// TIA Portal project "Energy_Monitoring_Project" (V17)

(* hardware
DEVICE "S7-1200 station_1"  S7-1200 Station
   slot 0: "Rack_0"  S7-1200 Rack  Rack  V1.0
   slot 1: "PLC_1"  CPU 1214C DC/DC/DC  6ES7 214-1AG40-0XB0  V4.5
DEVICE "HMI_1"  TP700 Comfort
   slot 0: "HMI_1"  TP700 Comfort  6AV2 124-0GC01-0AX0  17.0.0.0
   slot 1: "HMI_RT_1"  TP700 Comfort  6AV2 124-0GC01-0AX0  17.0.0.0
   slot 5: "HMI_1.IE_CP_1"  PROFINET Interface  17.0.0.0
      slot 1: "PROFINET Interface_1"  PROFINET Interface
         slot 1: "Port_1"  Port
         slot 2: "Port_2"  Port
   slot 7: "HMI_1.MPI/DP_CP_1"  MPI/DP Interface  17.0.0.0
*)

// ===== PLC "PLC_1"  CPU 1214C DC/DC/DC =====

VAR_GLOBAL   // PLC tag table "Default tag table"
   "Tag_1" AT %MW0 : Word;
   "Tag_2" AT %MW2 : Word;
   "Tag_3" AT %MW4 : Word;
   "Tag_4" AT %MW6 : Word;
   "Tag_5" AT %MW8 : Word;
   "Tag_6" AT %MW10 : Word;
   "Tag_7" AT %MW12 : Word;
   "Tag_8" AT %MW14 : Word;
   "Tag_9" AT %MW16 : Word;
END_VAR

DATA_BLOCK "Zone1_DB"   // DB1
{ S7_Optimized_Access := 'TRUE' }
VERSION : 0.1
   VAR
      Voltage : Real;
      Current : Real;
      kW : Real;
      kWh : Real;
      Threshold_Exceeded : Bool;
   END_VAR
BEGIN
END_DATA_BLOCK

DATA_BLOCK "Zone2_DB"   // DB2
{ S7_Optimized_Access := 'TRUE' }
VERSION : 0.1
   VAR
      Voltage : Real;
      Current : Real;
      kW : Real;
      kWh : Real;
      Threshold_Exceeded : Bool;
   END_VAR
BEGIN
END_DATA_BLOCK

DATA_BLOCK "Zone3_DB"   // DB3
{ S7_Optimized_Access := 'TRUE' }
VERSION : 0.1
   VAR
      Voltage : Real;
      Current : Real;
      kW : Real;
      kWh : Real;
      Threshold_Exceeded : Bool;
   END_VAR
BEGIN
END_DATA_BLOCK

DATA_BLOCK "Config_DB"   // DB4
{ S7_Optimized_Access := 'TRUE' }
VERSION : 0.1
   VAR
      Zone1_Threshold : Real := 50.0;   // Zone 1 max kW
      Zone2_Threshold : Real := 30.0;   // Zone 2 max kW
      Zone3_Threshold : Real := 20.0;   // Zone 3 max kW
      Total_Threshold : Real := 90.0;   // Total plant nax kW
      Shift_Start_Hour : Int := 8;   // Shift start time
      Alert_Enabled : Bool := true;   // Enable alerts
      Total_Power : Real;   // Total Power
      Shift_Number : Int := 1;
      Shift_Start_KWh : Real;
      Shift_Consumption : Real;
   END_VAR
BEGIN
END_DATA_BLOCK

DATA_BLOCK "Alarm_DB"   // DB5
{ S7_Optimized_Access := 'TRUE' }
VERSION : 0.1
   VAR
      Total_Exceeded : Bool;
      Alarm_Word : Word;
      Zone1_Alarm : Bool;
      Zone2_Alarm : Bool;
      Zone3_Alarm : Bool;
      Any_Alarm : Bool;
   END_VAR
BEGIN
END_DATA_BLOCK

DATA_BLOCK "Zone1_Reader_DB"   // DB6
{ S7_Optimized_Access := 'TRUE' }
VERSION : 0.1
// stored: InstanceOfName FB1_Energy_Reader
"FB1_Energy_Reader"
BEGIN
END_DATA_BLOCK

DATA_BLOCK "Zone2_Reader_DB"   // DB7
{ S7_Optimized_Access := 'TRUE' }
VERSION : 0.1
// stored: InstanceOfName FB1_Energy_Reader
"FB1_Energy_Reader"
BEGIN
END_DATA_BLOCK

DATA_BLOCK "Zone3_Reader_DB"   // DB8
{ S7_Optimized_Access := 'TRUE' }
VERSION : 0.1
// stored: InstanceOfName FB1_Energy_Reader
"FB1_Energy_Reader"
BEGIN
END_DATA_BLOCK

FUNCTION_BLOCK "FB1_Energy_Reader"   // FB1, SCL
{ S7_Optimized_Access := 'TRUE' }
VERSION : 0.1
   VAR_INPUT
      Voltage_Raw : Int;   // Raw analog voltage
      Current_Raw : Int;   // Raw analog current
      Power_Raw : Int;   // Raw analog power
      Zone_Name : String;   // Zone identifier
      Power_Threshold : Real;   // Alert thershold kW
   END_VAR
   VAR_OUTPUT
      Voltage : Real;   // Actual voltage V
      Current : Real;   // Actual Current A
      Active_Power : Real;   // Active Power kW
      Energy_kWh : Real;   // Cumulative energy
      Threshold_Exceeded : Bool;   // Alert flag
      Power_Factor : Real;   // PF calculation
   END_VAR
   VAR
      last_Power : Real;   // Previous scan power
      Scan_Timer : TON_TIME;   // 1 second timer
      kWh_Accumulator : Real;   // Running total
   END_VAR
BEGIN
   // --- Scale analog inputs ---
   #Voltage := INT_TO_REAL(#Voltage_Raw) / 27648.0 * 415.0;
   #Current := INT_TO_REAL(#Current_Raw) / 27648.0 * 100.0;
   #Active_Power := (#Voltage * #Current * #Power_Factor) / 1000.0;

   // --- Calculate kWh every second ---
   #Scan_Timer(IN := TRUE,
               PT := T#1S);

   IF #Scan_Timer.Q THEN
       #kWh_Accumulator := #kWh_Accumulator + (#Active_Power / 3600.0);
       #Scan_Timer(IN := FALSE,
                   PT := T#1S);
   END_IF;

   #Energy_kWh := #kWh_Accumulator;

   // --- Threshold check ---
   #Threshold_Exceeded := #Active_Power > #Power_Threshold;

   // --- Power factor (simplified) ---
   IF #Voltage > 0.0 AND #Current > 0.0 THEN
       #Power_Factor := 0.85; // Default - real system uses meter register
   END_IF;
END_FUNCTION_BLOCK

FUNCTION "FC1_Power_Calculation" : Void   // FC1, SCL
{ S7_Optimized_Access := 'TRUE' }
VERSION : 0.1
BEGIN
END_FUNCTION

FUNCTION "FC2_Alarm_generator" : Void   // FC2, SCL
{ S7_Optimized_Access := 'TRUE' }
VERSION : 0.1
   VAR_INPUT
      Zone1_Exceeded : Bool;
      Zone2_Exceeded : Bool;
      Zone3_Exceeded : Bool;
      Total_Exceeded : Bool;
   END_VAR
   VAR_OUTPUT
      Alarm_Word : Word;
      Any_Alarm : Bool;
   END_VAR
BEGIN
   // Pack alarms into word bits
   #Alarm_Word.%X0 := #Zone1_Exceeded;
   #Alarm_Word.%X1 := #Zone2_Exceeded;
   #Alarm_Word.%X2 := #Zone3_Exceeded;
   #Alarm_Word.%X3 := #Total_Exceeded;

   //Any alarm active
   #Any_Alarm := #Zone1_Exceeded OR
                 #Zone2_Exceeded OR
                 #Zone3_Exceeded OR
                 #Total_Exceeded;
END_FUNCTION

ORGANIZATION_BLOCK "Main"   // OB1, SCL, ProgramCycle
TITLE = "Main Program Sweep (Cycle)"
{ S7_Optimized_Access := 'TRUE' }
VERSION : 0.1
   VAR_INPUT
      Initial_Call : Bool;   // Initial call of this OB
      Remanence : Bool;   // =True, if remanent data are available
   END_VAR
BEGIN
   // ═══ ENERGY MONITORING SYSTEM ═══

   // Zone 1 — popup will ask to create Zone1_Reader_DB
   "Zone1_Reader_DB"(
                     Voltage_Raw     := "Tag_1",
                     Current_Raw     := "Tag_2",
                     Power_Raw       := "Tag_3",
                     Power_Threshold := "Config_DB".Zone1_Threshold);

   "Zone1_DB".kWh := "Zone1_Reader_DB".Energy_kWh;
   "Zone1_DB".kW := "Zone1_Reader_DB".Active_Power;

   // Zone 2
   "Zone2_Reader_DB"(
                     Voltage_Raw     := "Tag_4",
                     Current_Raw     := "Tag_5",
                     Power_Raw       := "Tag_6",
                     Power_Threshold := "Config_DB".Zone2_Threshold);

   "Zone2_DB".kWh := "Zone2_Reader_DB".Energy_kWh;
   "Zone2_DB".kW := "Zone2_Reader_DB".Active_Power;

   // Zone 3
   "Zone3_Reader_DB"(
                     Voltage_Raw     := "Tag_7",
                     Current_Raw     := "Tag_8",
                     Power_Raw       := "Tag_9",
                     Power_Threshold := "Config_DB".Zone3_Threshold);

   "Zone3_DB".kWh := "Zone3_Reader_DB".Energy_kWh;
   "Zone3_DB".kW := "Zone3_Reader_DB".Active_Power;

   // Total
   "Config_DB".Total_Power :=
   "Zone1_Reader_DB".Active_Power +
   "Zone2_Reader_DB".Active_Power +
   "Zone3_Reader_DB".Active_Power;

   "Alarm_DB".Total_Exceeded :=
   "Config_DB".Total_Power > "Config_DB".Total_Threshold;

   // -- Alarm Generator --
   "FC2_Alarm_generator"(Zone1_Exceeded:= "Zone1_Reader_DB".Threshold_Exceeded,
                         Zone2_Exceeded:= "Zone2_Reader_DB".Threshold_Exceeded,
                         Zone3_Exceeded:="Zone3_Reader_DB".Threshold_Exceeded,
                         Total_Exceeded:="Alarm_DB".Total_Exceeded,
                         Alarm_Word=>"Alarm_DB".Alarm_Word,
                         Any_Alarm=>"Alarm_DB".Any_Alarm);

   //Shift Consumption Tracker
   "Config_DB".Shift_Consumption :=
   "Zone1_Reader_DB".Energy_kWh +
   "Zone2_Reader_DB".Energy_kWh +
   "Zone3_Reader_DB".Energy_kWh -
   "Config_DB".Shift_Start_KWh;
END_ORGANIZATION_BLOCK

(* ===== HMI "HMI_RT_1" =====
system functions are stored by id; their names below are inferred from use
connection "HMI_Connection_1": ETHERNET, S7_1200_OMS

HMI tags "Default tag table"
   "Tag_ScreenNumber" : UInt, internal
   "Zone1_kW" : Real = PLC Zone1_Reader_DB.Active_Power, 1 s
   "Zone1_kWh" : Real = PLC Zone1_Reader_DB.Energy_kWh AT %DB1.DBD0, 1 s
   "Zone2_kW" : Real = PLC Zone2_Reader_DB.Active_Power AT %DB1.DBD0, 1 s
   "Zone2_kWh" : Real = PLC Zone2_Reader_DB.Energy_kWh AT %DB1.DBD0, 1 s
   "Zone3_kW" : Real = PLC Zone3_Reader_DB.Active_Power AT %DB1.DBD0, 1 s
   "Zone3_kWh" : Real = PLC Zone3_Reader_DB.Energy_kWh AT %DB1.DBD0, 1 s
   "Total_kW" : Real = PLC Config_DB.Total_Power AT %DB1.DBD0, 1 s
   "Zone1_Alert" : Bool = PLC Zone1_Reader_DB.Threshold_Exceeded AT %DB1.DBX0.0, 1 s
   "Zone2_Alert" : Bool = PLC Zone2_Reader_DB.Threshold_Exceeded AT %DB1.DBX0.0, 1 s
   "Zone3_Alert" : Bool = PLC Zone3_Reader_DB.Threshold_Exceeded AT %DB1.DBX0.0, 1 s
   "Alarm_Active" : Bool = PLC Alarm_DB.Any_Alarm AT %DB1.DBX0.0, 1 s
   "Alarm_Word" : Word = PLC Alarm_DB.Alarm_Word AT %DB1.DBX0.0, 1 s

discrete alarms
   1: '', class Errors, trigger "Alarm_Word" bit 0
   2: '', class Errors, trigger "Alarm_Word" bit 1
   3: '', class Errors, trigger "Alarm_Word" bit 2
   4: '', class Errors, trigger "Alarm_Word" bit 3

screen "Root screen" 800x420, template "Template_1"
   on GenerateScreen: SetTag("Tag_ScreenNumber", 1)
   Visibility <- "Alarm_Active"
   IOField "I/O field_1" at 279,28 size 78x32; FormatPattern 999.9
      ProcessValue <- "Total_kW"
   TextField "Text field_1" at 72,33 size 216x23; Text 'TOTAL PLANT POWER:'
   TextField "Text field_2" at 364,33 size 33x23; Text 'kW'
   IOField "I/O field_2" at 159,76 size 58x32; FormatPattern 99.9
      ProcessValue <- "Zone1_kW"
   TextField "Text field_3" at 72,81 size 77x23; Text 'ZONE 1:'
   TextField "Text field_4" at 220,81 size 46x23; Text 'kW'
   IOField "I/O field_3" at 159,116 size 78x32; FormatPattern 9999.9
      ProcessValue <- "Zone1_kWh"
   TextField "Text field_5" at 244,121 size 44x23; Text 'kWh'
   Bar "Bar_1" at 160,159 size 88x54; MinimumValue 0; MaximumValue 50
      ProcessValue <- "Zone1_kW"
   Circle "Circle_1" at 167,232 size 48x48
      Appearance <- "Zone1_Alert"
   TextField "Text field_6" at 131,291 size 247x23; Text '⚠ THRESHOLD EXCEEDED!'
   IOField "I/O field_4" at 391,76 size 54x32; FormatPattern 99.9
      ProcessValue <- "Zone2_kW"
   TextField "Text field_7" at 304,81 size 77x23; Text 'ZONE 2:'
   TextField "Text field_8" at 455,81 size 38x23; Text 'kW'
   IOField "I/O field_5" at 391,116 size 78x32; FormatPattern 9999.9
      ProcessValue <- "Zone2_kWh"
   TextField "Text field_9" at 476,121 size 44x23; Text 'kWh'
   Bar "Bar_2" at 388,161 size 105x54; MinimumValue 0; MaximumValue 50
      ProcessValue <- "Zone2_kW"
   Circle "Circle_2" at 391,231 size 48x48
      Appearance <- "Zone2_Alert"
   IOField "I/O field_6" at 607,76 size 58x32; FormatPattern 99.9
      ProcessValue <- "Zone3_kW"
   TextField "Text field_10" at 536,81 size 77x23; Text 'ZONE 3:'
   TextField "Text field_11" at 676,81 size 41x23; Text 'kW'
   IOField "I/O field_7" at 607,116 size 78x32; FormatPattern 9999.9
      ProcessValue <- "Zone3_kWh"
   TextField "Text field_12" at 692,121 size 53x23; Text 'kWh'
   Bar "Bar_3" at 606,161 size 103x54; MinimumValue 0; MaximumValue 50
      ProcessValue <- "Zone3_kW"
   Circle "Circle_3" at 615,232 size 48x48
      Appearance <- "Zone3_Alert"
   Button "Button_1" at 643,367 size 71x47; TextOff 'Trends'
      on Press: ActivateScreen("Energy_Trends", 0)
   Button "Button_2" at 563,367 size 71x47; TextOff 'Alarms'
      on Press: ActivateScreen("Alarm_Screen", 0)

Template "Template_1" 800x420
   Button "Exit" at 720,360 size 78x58; TextOff 'Exit'; PictureOff "ExitRuntime_TP700_Comfort_TR"; PictureOn "ExitRuntime_TP700_Comfort_TR"
      on Release: StopRuntime(0)
   Button "Template_Button" at 640,360 size 78x58; TextOff 'Text'
   Button "Template_Button_1" at 560,360 size 78x58; TextOff 'Text'
   Button "Template_Button_2" at 480,360 size 78x58; TextOff 'Text'
   Button "Template_Button_3" at 400,360 size 78x58; TextOff 'Text'
   Button "Template_Button_4" at 321,360 size 78x58; TextOff 'Text'
   Button "Template_Button_5" at 241,360 size 78x58; TextOff 'Text'
   Button "Template_Button_6" at 161,360 size 78x58; TextOff 'Text'
   Button "Alarms" at 81,360 size 78x58; TextOff 'Alarms'; PictureOff "AlarmDisplay_TP700_Comfort_TR"; PictureOn "AlarmDisplay_TP700_Comfort_TR"
      on Release: function_ef3f5d25("Alarm window_Unacknowledged", -1)
   Button "Start screen" at 1,360 size 78x58; TextOff 'Start screen'; PictureOff "NavigateHome_TP700_Comfort_TR"; PictureOn "NavigateHome_TP700_Comfort_TR"
      on Release: ActivateScreen("Root screen", 0)

screen "Energy_Trends" 800x420
   TrendView "Trend view_1" at 9,0 size 688x405
   Button "Button_2" at 714,362 size 71x47; TextOff 'Back'
      on Click: ActivateScreen("Root screen", 0)

screen "Alarm_Screen" 800x420
   AlarmView "Alarm view_1" at 23,4 size 708x300
   Button "Button_2" at 714,362 size 71x47; TextOff 'Back'
      on Click: ActivateScreen("Screen_1", 0)

screen "Screen_1" 800x420
   TextField "Text field_3" at 72,81 size 77x23; Text 'ZONE 1:'
   TextField "Text field_4" at 220,81 size 41x23; Text 'kW'
   IOField "I/O field_3" at 156,116 size 78x32; FormatPattern 9999.9
      ProcessValue <- "Zone1_kWh"
   TextField "Text field_5" at 236,121 size 47x21; Text 'kWh'
   Bar "Bar_1" at 156,159 size 104x54; MinimumValue 0; MaximumValue 50
      ProcessValue <- "Zone1_kW"
   Circle "Circle_1" at 156,232 size 48x48
      Appearance <- "Zone1_Alert"
   IOField "I/O field_1" at 287,28 size 68x32; FormatPattern 999.9
      ProcessValue <- "Total_kW"
   TextField "Text field_1" at 72,33 size 216x23; Text 'TOTAL PLANT POWER:'
   TextField "Text field_2" at 356,33 size 42x23; Text 'kW'
   IOField "I/O field_2" at 156,76 size 56x32; FormatPattern 99.9
      ProcessValue <- "Zone1_kW"
   TextField "Text field_6" at 320,81 size 77x23; Text 'ZONE 2:'
   TextField "Text field_7" at 552,81 size 77x23; Text 'ZONE 3:'
   IOField "I/O field_4" at 391,76 size 54x32; FormatPattern 99.9
      ProcessValue <- "Zone2_kW"
   TextField "Text field_8" at 455,81 size 38x23; Text 'kW'
   IOField "I/O field_5" at 391,116 size 78x32; FormatPattern 9999.9
      ProcessValue <- "Zone2_kWh"
   TextField "Text field_9" at 476,121 size 44x23; Text 'kWh'
   Circle "Circle_2" at 391,231 size 48x48
      Appearance <- "Zone2_Alert"
   Bar "Bar_2" at 388,159 size 104x54; MinimumValue 0; MaximumValue 50
      ProcessValue <- "Zone2_kW"
   IOField "I/O field_6" at 623,76 size 58x32; FormatPattern 99.9
      ProcessValue <- "Zone3_kW"
   IOField "I/O field_7" at 623,116 size 78x32; FormatPattern 9999.9
      ProcessValue <- "Zone3_kWh"
   Circle "Circle_3" at 631,232 size 48x48
      Appearance <- "Zone3_Alert"
   TextField "Text field_10" at 687,81 size 38x23; Text 'kW'
   TextField "Text field_11" at 708,121 size 44x23; Text 'kWh'
   Bar "Bar_3" at 612,159 size 104x54; MinimumValue 0; MaximumValue 50
      ProcessValue <- "Zone3_kW"
   TextField "Text field_12" at 131,291 size 247x23; Text '⚠ THRESHOLD EXCEEDED!'
   Button "Button_1" at 643,367 size 71x47; TextOff 'Trends'
      on Press: ActivateScreen("Energy_Trends", 0)
   Button "Button_2" at 563,367 size 71x47; TextOff 'Alarms'
      on Press: ActivateScreen("Alarm_Screen", 0)
*)